(* IEC 61131-3 sources: ae-demo-rack/src, 3 files *)

(* ---- vplc-427e_IoAddresses.st ---- *)
CONFIGURATION IoAddresses
    VAR_GLOBAL

        // Module device_drive_center_s200/drivespd
        device_drive_center_s200_drivespd_Input AT %IB288 : device_drive_center_s200_drivespd_Input_Layout;
        device_drive_center_s200_drivespd_Output AT %QB288 : device_drive_center_s200_drivespd_Output_Layout;

        // Module device_drive_left_s200/drivespd
        device_drive_left_s200_drivespd_Input AT %IB256 : device_drive_left_s200_drivespd_Input_Layout;
        device_drive_left_s200_drivespd_Output AT %QB256 : device_drive_left_s200_drivespd_Output_Layout;

        // Module device_drive_right_s200/drivespd
        device_drive_right_s200_drivespd_Input AT %IB320 : device_drive_right_s200_drivespd_Input_Layout;
        device_drive_right_s200_drivespd_Output AT %QB320 : device_drive_right_s200_drivespd_Output_Layout;

        // Module device_et200sp/ai4_1
        device_et200sp_ai4_1_Input AT %IB0 : device_et200sp_ai4_1_Input_Layout;

        // Module device_et200sp/di8_1
        io_switch_board_lc_s AT %IB9 : device_et200sp_di8_1_Input_Layout;

        // Module device_et200sp/di8_2
        io_switch_board_cr AT %IB8 : device_et200sp_di8_2_Input_Layout;

        // Module device_et200sp/dq8_1
        io_led_board_lc AT %QB1 : device_et200sp_dq8_1_Output_Layout;

        // Module device_et200sp/dq8_2
        io_led_board_cr AT %QB0 : device_et200sp_dq8_2_Output_Layout;
    END_VAR
END_CONFIGURATION

TYPE
    device_drive_center_s200_drivespd_Input_Layout : STRUCT
        Signals_0 AT %B0 : WORD;
        Signals_1 AT %B2 : WORD;
    END_STRUCT;
END_TYPE

TYPE
    device_drive_center_s200_drivespd_Output_Layout : STRUCT
        Signals_2 AT %B0 : WORD;
        Signals_3 AT %B2 : WORD;
    END_STRUCT;
END_TYPE

TYPE
    device_drive_left_s200_drivespd_Input_Layout : STRUCT
        Signals_0 AT %B0 : WORD;
        Signals_1 AT %B2 : WORD;
    END_STRUCT;
END_TYPE

TYPE
    device_drive_left_s200_drivespd_Output_Layout : STRUCT
        Signals_2 AT %B0 : WORD;
        Signals_3 AT %B2 : WORD;
    END_STRUCT;
END_TYPE

TYPE
    device_drive_right_s200_drivespd_Input_Layout : STRUCT
        Signals_0 AT %B0 : WORD;
        Signals_1 AT %B2 : WORD;
    END_STRUCT;
END_TYPE

TYPE
    device_drive_right_s200_drivespd_Output_Layout : STRUCT
        Signals_2 AT %B0 : WORD;
        Signals_3 AT %B2 : WORD;
    END_STRUCT;
END_TYPE

TYPE
    device_et200sp_ai4_1_Input_Layout : STRUCT
        Signals_0 AT %B0 : INT;
        Signals_1 AT %B2 : INT;
        Signals_2 AT %B4 : INT;
        Signals_3 AT %B6 : INT;
    END_STRUCT;
END_TYPE

TYPE
    device_et200sp_di8_1_Input_Layout : STRUCT
        switchleft0 AT %X0.0 : BOOL;
        switchleft1 AT %X0.1 : BOOL;
        switchleft2 AT %X0.2 : BOOL;
        switchleft3 AT %X0.3 : BOOL;
        switchcenter0 AT %X0.4 : BOOL;
        switchcenter1 AT %X0.5 : BOOL;
        estop AT %X0.6 : BOOL;
        Signals_7 AT %X0.7 : BOOL;
    END_STRUCT;
END_TYPE

TYPE
    device_et200sp_di8_2_Input_Layout : STRUCT
        switchcenter2 AT %X0.0 : BOOL;
        switchcenter3 AT %X0.1 : BOOL;
        switchright0 AT %X0.2 : BOOL;
        switchright1 AT %X0.3 : BOOL;
        switchright2 AT %X0.4 : BOOL;
        switchright3 AT %X0.5 : BOOL;
        Signals_6 AT %X0.6 : BOOL;
        Signals_7 AT %X0.7 : BOOL;
    END_STRUCT;
END_TYPE

TYPE
    device_et200sp_dq8_1_Output_Layout : STRUCT
        ledleft0 AT %X0.0 : BOOL;
        ledleft1 AT %X0.1 : BOOL;
        ledleft2 AT %X0.2 : BOOL;
        ledleft3 AT %X0.3 : BOOL;
        ledcenter0 AT %X0.4 : BOOL;
        ledcenter1 AT %X0.5 : BOOL;
        Signals_6 AT %X0.6 : BOOL;
        Signals_7 AT %X0.7 : BOOL;
    END_STRUCT;
END_TYPE

TYPE
    device_et200sp_dq8_2_Output_Layout : STRUCT
        ledcenter2 AT %X0.0 : BOOL;
        ledcenter3 AT %X0.1 : BOOL;
        ledright0 AT %X0.2 : BOOL;
        ledright1 AT %X0.3 : BOOL;
        ledright2 AT %X0.4 : BOOL;
        ledright3 AT %X0.5 : BOOL;
        Signals_6 AT %X0.6 : BOOL;
        Signals_7 AT %X0.7 : BOOL;
    END_STRUCT;
END_TYPE

(* ---- vplc-427e_HwIdentifiers.st ---- *)
CONFIGURATION HardwareIDs
    VAR_GLOBAL CONSTANT
        device_drive_center_s200_HwID : UINT := UINT#282;
        device_drive_center_s200_Rack_HwID : UINT := UINT#285;
        device_drive_center_s200_drivespd_HwID : UINT := UINT#287;
        device_drive_center_s200_drivespd_Module_Access_Point_HwID : UINT := UINT#289;
        device_drive_center_s200_drivespd_leeres_Submodul_HwID : UINT := UINT#288;
        device_drive_center_s200_s200_center_HwID : UINT := UINT#286;
        device_drive_center_s200_s200_center_PN_IO_HwID : UINT := UINT#281;
        device_drive_center_s200_s200_center_PN_IO_Port_1_HwID : UINT := UINT#283;
        device_drive_center_s200_s200_center_PN_IO_Port_2_HwID : UINT := UINT#284;
        device_drive_center_s200_s200_center_SINAMICS_S200_PN_V6_4_HwID : UINT := UINT#291;
        device_drive_center_s200_telegram1_HwID : UINT := UINT#290;
        device_drive_left_s200_HwID : UINT := UINT#293;
        device_drive_left_s200_Rack_HwID : UINT := UINT#296;
        device_drive_left_s200_drivespd_HwID : UINT := UINT#298;
        device_drive_left_s200_drivespd_Module_Access_Point_HwID : UINT := UINT#301;
        device_drive_left_s200_drivespd_leeres_Submodul_HwID : UINT := UINT#299;
        device_drive_left_s200_s200_left_HwID : UINT := UINT#297;
        device_drive_left_s200_s200_left_PN_IO_HwID : UINT := UINT#292;
        device_drive_left_s200_s200_left_PN_IO_Port_1_HwID : UINT := UINT#294;
        device_drive_left_s200_s200_left_PN_IO_Port_2_HwID : UINT := UINT#295;
        device_drive_left_s200_s200_left_SINAMICS_S200_PN_V6_4_HwID : UINT := UINT#303;
        device_drive_left_s200_telegram1_HwID : UINT := UINT#302;
        device_drive_right_s200_HwID : UINT := UINT#271;
        device_drive_right_s200_Rack_HwID : UINT := UINT#274;
        device_drive_right_s200_drivespd_HwID : UINT := UINT#276;
        device_drive_right_s200_drivespd_Module_Access_Point_HwID : UINT := UINT#278;
        device_drive_right_s200_drivespd_leeres_Submodul_HwID : UINT := UINT#277;
        device_drive_right_s200_s200_right_HwID : UINT := UINT#275;
        device_drive_right_s200_s200_right_PN_IO_HwID : UINT := UINT#270;
        device_drive_right_s200_s200_right_PN_IO_Port_1_HwID : UINT := UINT#272;
        device_drive_right_s200_s200_right_PN_IO_Port_2_HwID : UINT := UINT#273;
        device_drive_right_s200_s200_right_SINAMICS_S200_PN_V6_4_HwID : UINT := UINT#280;
        device_drive_right_s200_telegram1_HwID : UINT := UINT#279;
        device_et200sp_HwID : UINT := UINT#258;
        device_et200sp_Rack_HwID : UINT := UINT#261;
        device_et200sp_ai4_1_AI_4xI_2__4_wire_ST_V2_0_HwID : UINT := UINT#264;
        device_et200sp_di8_1_DI_8x24VDC_HF_V2_0_HwID : UINT := UINT#268;
        device_et200sp_di8_2_DI_8x24VDC_HS_V1_0_HwID : UINT := UINT#267;
        device_et200sp_dq8_1_DQ_8x24VDC_0_5A_HF_V2_0_HwID : UINT := UINT#266;
        device_et200sp_dq8_2_DQ_8x24VDC_0_5A_ST_V0_0_HwID : UINT := UINT#265;
        device_et200sp_im_155_6_HwID : UINT := UINT#262;
        device_et200sp_im_155_6_IM_155_6_PN_2_HF_V4_2_HwID : UINT := UINT#269;
        device_et200sp_im_155_6_PN_IO_HwID : UINT := UINT#257;
        device_et200sp_im_155_6_Port_1_HwID : UINT := UINT#259;
        device_et200sp_im_155_6_Port_2_HwID : UINT := UINT#260;
        device_et200sp_server_mod_Servermodul_V1_1_0_Bytes_HwID : UINT := UINT#263;
        device_plc_HwID : UINT := UINT#32;
        device_plc_Rail_0_HwID : UINT := UINT#300;
        device_plc_vplc_427e_HwID : UINT := UINT#48;
        device_plc_vplc_427e_Card_reader_writer_1_HwID : UINT := UINT#51;
        device_plc_vplc_427e_OPC_UA_1_HwID : UINT := UINT#117;
        device_plc_vplc_427e_PROFINET_interface_1_HwID : UINT := UINT#64;
        device_plc_vplc_427e_PROFINET_interface_1_Port_1_HwID : UINT := UINT#65;
        profinet_io_system_HwID : UINT := UINT#256;

    END_VAR
END_CONFIGURATION

(* ---- configuration.st ---- *)
CONFIGURATION ConfigurationRack

    TASK Main(Priority := 1);
    PROGRAM P1 WITH Main : ConsoleProgram;

    // >>> Global Variables
    {S7.Extern = ReadWrite}
    {OpcUa.AccessLevel = ReadWrite}
    VAR_GLOBAL
        driveLeftSpeedIncrease : INT := SPEED_INCREASE_DEFAULT;
        driveCenterSpeedIncrease : INT  := SPEED_INCREASE_DEFAULT;
        driveRightSpeedIncrease : INT  := SPEED_INCREASE_DEFAULT;
    END_VAR

    {S7.Extern = ReadOnly}
    {OpcUa.AccessLevel = ReadOnly}
    VAR_GLOBAL
        estopActive : BOOL;
        driveLeftActive : BOOL;
        driveLeftTargetSpeed : LREAL; // := SPEED_INITIAL;
        driveCenterActive : BOOL;
        driveCenterTargetSpeed : LREAL; // := SPEED_INITIAL;
        driveRightActive : BOOL;
        driveRightTargetSpeed : LREAL; // := SPEED_INITIAL;
    END_VAR

    // >>> Global IO-Tags
    VAR_GLOBAL
        // see : vplc-427e_IoAddresses.st
    END_VAR

    // >>> Global Constants
    VAR_GLOBAL CONSTANT
        SPEED_INCREASE_DEFAULT : INT := 10;
        SPEED_INITIAL : LREAL := LREAL#100.0;
    END_VAR

END_CONFIGURATION
